FUNCTION f_XpuOperationModeToString : string(30)
VAR_INPUT
  nOperationMode    : uint;
END_VAR
VAR
END_VAR


CASE nOperationMode
OF
  0:
    f_XpuOperationModeToString    := 'Normal';

  1:
    f_XpuOperationModeToString    := 'Simulation';
ELSE
    f_XpuOperationModeToString    := 'UNKNOWN OP mode';
END_CASE

END_FUNCTION

(* stored: Version 1.1.0.1, ProductVersion 3.1.4024.12
   POU f_XpuOperationModeToString: Id {ee065be4-8c4f-4c98-9163-f7f845304857}, SpecialFunc None *)
